// TwinCAT 3 PLC project Conveyor11
// ProgramVersion: 3.1.4026.10
// CompilerDefines: VISU_USEPROPERTYINFO
// libraries:
//   Tc2_Standard, * (Beckhoff Automation GmbH)
//   Tc2_System, * (Beckhoff Automation GmbH)
// project tree:
//   / GlobalTextList.TcGTLO, PlcTask.TcTTO, Visualization Manager.TcVMO (not stored)
//   GVLs/ GVL.TcGVL
//   POUs/ MAIN.TcPOU, Simulation.TcPOU
//   VISUs/ Visualization.TcVIS
// real-time tasks:
//   TASK PlcTask: cycle T#10ms, priority 20, ADS port 350

CONFIGURATION Conveyor11
    RESOURCE PLC ON TwinCAT3
        TASK PlcTask(INTERVAL := T#10ms, PRIORITY := 20);
        PROGRAM Simulation WITH PlcTask : Simulation;
        PROGRAM MAIN WITH PlcTask : MAIN;
    END_RESOURCE
END_CONFIGURATION

// ---- GVLs/GVL.TcGVL
{attribute 'qualified_only'}
VAR_GLOBAL
	_MotorOnOff				:BOOL;
	_SensorCovered			:BOOL;
	_Switch					:BOOL;
	_PackageIsPlaced		:BOOL;
	_RetainedTimeOnConveyor	:TIME;
	_MovementTime			:TIME := T#10S;		//How long it takes for the package to move through the conveyor
END_VAR

// ---- POUs/Simulation.TcPOU
PROGRAM Simulation
VAR
	_ConveyorTimer		:TON;				//Where in the conveyor is the package
	_TimeOnConveyor		:TIME;
END_VAR


//This program simulates the conveyor's movement, which is represented as a bar in the visualisation.
//Placing of a package on the conveyor is represented with a variable, and that's when the timer starts.
//If the conveyor is stopped while the package moves, the value for it's location must be retained (in
//this case the time value is retained).

IF GVL._MotorOnOff AND GVL._PackageIsPlaced THEN
	_ConveyorTimer(IN:= GVL._PackageIsPlaced, PT:= (GVL._MovementTime-_TimeOnConveyor), Q=> GVL._SensorCovered, ET=> _TimeOnConveyor);
	IF GVL._SensorCovered THEN
		GVL._MotorOnOff := FALSE;
	ELSIF NOT GVL._SensorCovered AND GVL._PackageIsPlaced THEN
		_TimeOnConveyor := GVL._RetainedTimeOnConveyor;
	END_IF
END_IF

END_PROGRAM

// ---- POUs/MAIN.TcPOU
PROGRAM MAIN
VAR
END_VAR

IF NOT GVL._SensorCovered AND GVL._Switch THEN
	GVL._MotorOnOff := TRUE;
ELSE
	GVL._MotorOnOff := FALSE;
END_IF

END_PROGRAM

// ---- GlobalTextList.TcGTLO
TEXTLIST GlobalTextList
  854 = 'B1'
  461 = 'Motor M1 On/Off'
END_TEXTLIST

// ---- VISUs/Visualization.TcVIS
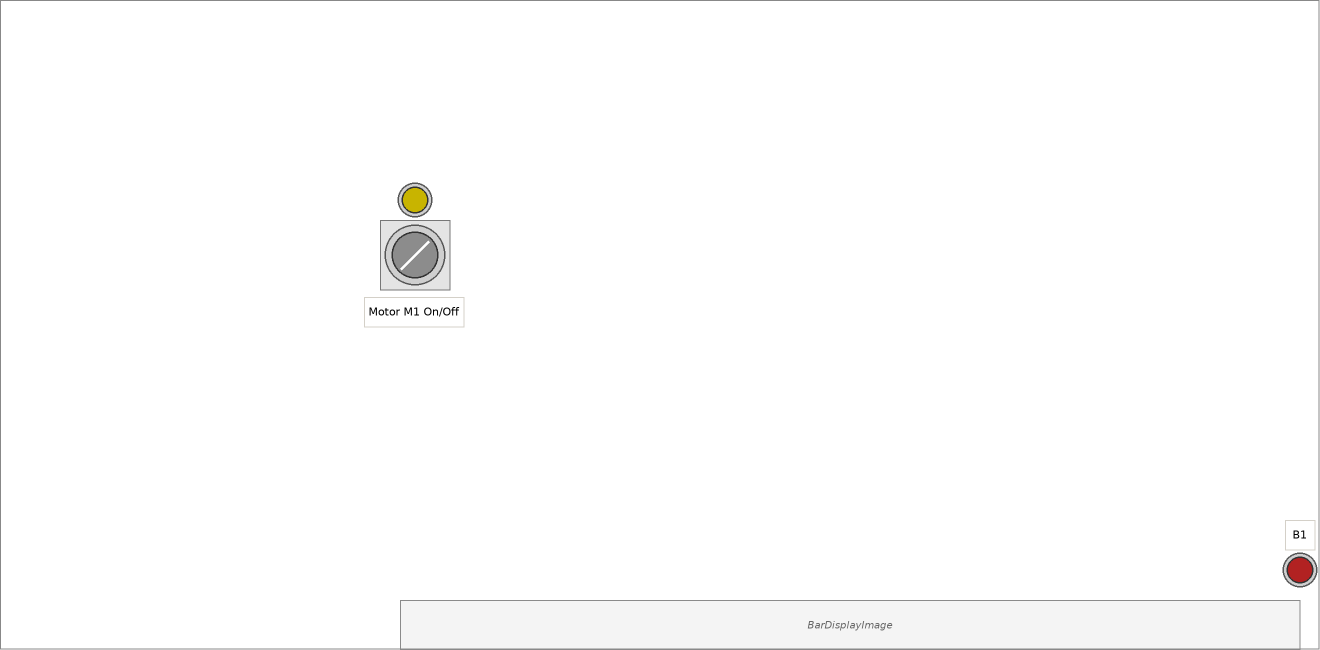
VISUALIZATION Visualization  // 1320x650
VAR_IN_OUT
END_VAR
//Palkki ei liiku, lisää napit paketin laittamiselle ja poistamiselle
    BarDisplayImage (400,600 900x50), value: GVL._TimeOnConveyor, style: BarDisplayImage-Blue, scale format: %.1f, scale 0..100
    RotarySwitch (380,220 70x70), variable: GVL._Switch, behaviour: TOGGLE, style: Switch-RotarySwitch-Gray
    Lamp1 (1280,550 40x40), variable: GVL._SensorCovered, style: Lamp-Lamp1-Red
    Textfield (1285,520 30x30), "B1"
    Textfield (364,297 100x30), "Motor M1 On/Off"
    Lamp1 (395,180 40x40), variable: GVL._Switch, style: Lamp-Lamp1-Yellow
END_VISUALIZATION
